Staubli VAL3: primeAreaTest.pgx

public program primeAreaTest()
begin
  // reset test state machine
  nAreaTestState=0
end
